ABB RAPID module: Module1.mod

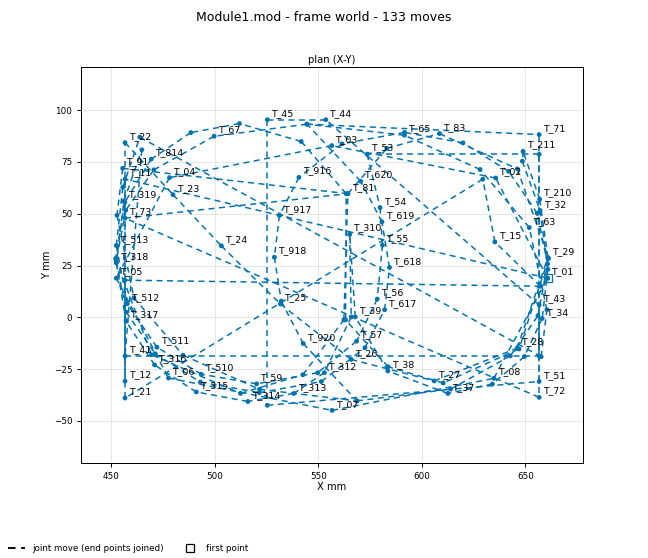
[picture p0: tool path of Module1.mod in frame world, 133 of 133 moves have a stored position in this frame; points joined in program order, loops and branches not executed]
MODULE Module1
    TASK PERS wobjdata Workobject_1:=[FALSE,TRUE,"",[[350,-300,410],[0,0,1,0]],[[0,0,0],[1,0,0,0]]];
    !Zero points
    CONST robtarget T_01:=[[-310.742,318.894,0],[1,0,0,0],[0,0,0,0],[9E+09,9E+09,9E+09,9E+09,9E+09,9E+09]];
    CONST robtarget T_02:=[[-285.702,367.273,0],[1,0,0,0],[0,0,0,0],[9E+09,9E+09,9E+09,9E+09,9E+09,9E+09]];
    CONST robtarget T_03:=[[-206.529,382.913,0],[1,0,0,0],[0,0,0,0],[9E+09,9E+09,9E+09,9E+09,9E+09,9E+09]];
    CONST robtarget T_04:=[[-128.165,367.435,0],[1,0,0,0],[0,0,0,0],[9E+09,9E+09,9E+09,9E+09,9E+09,9E+09]];
    CONST robtarget T_05:=[[-102.477,318.894,0],[1,0,0,0],[0,0,0,0],[9E+09,9E+09,9E+09,9E+09,9E+09,9E+09]];
    CONST robtarget T_06:=[[-127.679,270.676,0],[1,0,0,0],[0,0,0,0],[9E+09,9E+09,9E+09,9E+09,9E+09,9E+09]];
    CONST robtarget T_07:=[[-206.691,255.036,0],[1,0,0,0],[0,0,0,0],[9E+09,9E+09,9E+09,9E+09,9E+09,9E+09]];
    CONST robtarget T_08:=[[-284.811,270.514,0],[1,0,0,0],[0,0,0,0],[9E+09,9E+09,9E+09,9E+09,9E+09,9E+09]];
    CONST robtarget T_09:=[[-310.742,318.894,0],[1,0,0,0],[0,0,0,0],[9E+09,9E+09,9E+09,9E+09,9E+09,9E+09]];
    !One points
    CONST robtarget T_11:=[[-106.691,366.707,0],[1,0,0,0],[0,0,0,0],[9E+09,9E+09,9E+09,9E+09,9E+09,9E+09]];
    CONST robtarget T_12:=[[-106.691,269.138,0],[1,0,0,0],[0,0,0,0],[9E+09,9E+09,9E+09,9E+09,9E+09,9E+09]];
    CONST robtarget T_13:=[[-106.691,317.923,0],[1,0,0,0],[0,0,0,0],[9E+09,9E+09,9E+09,9E+09,9E+09,9E+09]];
    CONST robtarget T_14:=[[-307.339,315.005,0],[1,0,0,0],[0,0,0,0],[9E+09,9E+09,9E+09,9E+09,9E+09,9E+09]];
    CONST robtarget T_15:=[[-285.297,336.399,0],[1,0,0,0],[0,0,0,0],[9E+09,9E+09,9E+09,9E+09,9E+09,9E+09]];
    CONST robtarget T_16:=[[-279.462,366.707,0],[1,0,0,0],[0,0,0,0],[9E+09,9E+09,9E+09,9E+09,9E+09,9E+09]];
    !Two points
    CONST robtarget T_21:=[[-106.691,261.009,0],[1,0,0,0],[0,0,0,0],[9E+09,9E+09,9E+09,9E+09,9E+09,9E+09]];
    CONST robtarget T_22:=[[-106.691,384.347,0],[1,0,0,0],[0,0,0,0],[9E+09,9E+09,9E+09,9E+09,9E+09,9E+09]];
    CONST robtarget T_23:=[[-129.867,359.226,0],[1,0,0,0],[0,0,0,0],[9E+09,9E+09,9E+09,9E+09,9E+09,9E+09]];
    CONST robtarget T_24:=[[-153.206,334.509,0],[1,0,0,0],[0,0,0,0],[9E+09,9E+09,9E+09,9E+09,9E+09,9E+09]];
    CONST robtarget T_25:=[[-181.731,306.39,0],[1,0,0,0],[0,0,0,0],[9E+09,9E+09,9E+09,9E+09,9E+09,9E+09]];
    CONST robtarget T_26:=[[-215.929,279.647,0],[1,0,0,0],[0,0,0,0],[9E+09,9E+09,9E+09,9E+09,9E+09,9E+09]];
    CONST robtarget T_27:=[[-255.961,269.274,0],[1,0,0,0],[0,0,0,0],[9E+09,9E+09,9E+09,9E+09,9E+09,9E+09]];
    CONST robtarget T_28:=[[-296.075,285.077,0],[1,0,0,0],[0,0,0,0],[9E+09,9E+09,9E+09,9E+09,9E+09,9E+09]];
    CONST robtarget T_29:=[[-310.905,328.918,0],[1,0,0,0],[0,0,0,0],[9E+09,9E+09,9E+09,9E+09,9E+09,9E+09]];
    CONST robtarget T_210:=[[-306.934,357.038,0],[1,0,0,0],[0,0,0,0],[9E+09,9E+09,9E+09,9E+09,9E+09,9E+09]];
    CONST robtarget T_211:=[[-298.911,380.133,0],[1,0,0,0],[0,0,0,0],[9E+09,9E+09,9E+09,9E+09,9E+09,9E+09]];
    !Three points
    CONST robtarget T_31:=[[-298.587,375.377,0],[1,0,0,0],[0,0,0,0],[9E+09,9E+09,9E+09,9E+09,9E+09,9E+09]];
    CONST robtarget T_32:=[[-307.096,351.633,0],[1,0,0,0],[0,0,0,0],[9E+09,9E+09,9E+09,9E+09,9E+09,9E+09]];
    CONST robtarget T_33:=[[-310.905,323.189,0],[1,0,0,0],[0,0,0,0],[9E+09,9E+09,9E+09,9E+09,9E+09,9E+09]];
    CONST robtarget T_34:=[[-308.149,299.445,0],[1,0,0,0],[0,0,0,0],[9E+09,9E+09,9E+09,9E+09,9E+09,9E+09]];
    CONST robtarget T_35:=[[-299.559,281.049,0],[1,0,0,0],[0,0,0,0],[9E+09,9E+09,9E+09,9E+09,9E+09,9E+09]];
    CONST robtarget T_36:=[[-284.081,267.759,0],[1,0,0,0],[0,0,0,0],[9E+09,9E+09,9E+09,9E+09,9E+09,9E+09]];
    CONST robtarget T_37:=[[-262.606,263.221,0],[1,0,0,0],[0,0,0,0],[9E+09,9E+09,9E+09,9E+09,9E+09,9E+09]];
    CONST robtarget T_38:=[[-233.595,274.08,0],[1,0,0,0],[0,0,0,0],[9E+09,9E+09,9E+09,9E+09,9E+09,9E+09]];
    CONST robtarget T_39:=[[-217.874,300.174,0],[1,0,0,0],[0,0,0,0],[9E+09,9E+09,9E+09,9E+09,9E+09,9E+09]];
    CONST robtarget T_310:=[[-215.199,340.044,0],[1,0,0,0],[0,0,0,0],[9E+09,9E+09,9E+09,9E+09,9E+09,9E+09]];
    CONST robtarget T_311:=[[-215.929,300.174,0],[1,0,0,0],[0,0,0,0],[9E+09,9E+09,9E+09,9E+09,9E+09,9E+09]];
    CONST robtarget T_312:=[[-202.963,273.27,0],[1,0,0,0],[0,0,0,0],[9E+09,9E+09,9E+09,9E+09,9E+09,9E+09]];
    CONST robtarget T_313:=[[-188.214,263.221,0],[1,0,0,0],[0,0,0,0],[9E+09,9E+09,9E+09,9E+09,9E+09,9E+09]];
    CONST robtarget T_314:=[[-166.01,259.331,0],[1,0,0,0],[0,0,0,0],[9E+09,9E+09,9E+09,9E+09,9E+09,9E+09]];
    CONST robtarget T_315:=[[-141.131,263.95,0],[1,0,0,0],[0,0,0,0],[9E+09,9E+09,9E+09,9E+09,9E+09,9E+09]];
    CONST robtarget T_316:=[[-120.953,276.997,0],[1,0,0,0],[0,0,0,0],[9E+09,9E+09,9E+09,9E+09,9E+09,9E+09]];
    CONST robtarget T_317:=[[-107.177,298.148,0],[1,0,0,0],[0,0,0,0],[9E+09,9E+09,9E+09,9E+09,9E+09,9E+09]];
    CONST robtarget T_318:=[[-102.477,326.268,0],[1,0,0,0],[0,0,0,0],[9E+09,9E+09,9E+09,9E+09,9E+09,9E+09]];
    CONST robtarget T_319:=[[-106.123,356.09,0],[1,0,0,0],[0,0,0,0],[9E+09,9E+09,9E+09,9E+09,9E+09,9E+09]];
    CONST robtarget T_320:=[[-114.794,380.887,0],[1,0,0,0],[0,0,0,0],[9E+09,9E+09,9E+09,9E+09,9E+09,9E+09]];
    !Four points
    CONST robtarget T_41:=[[-106.691,281.323,0],[1,0,0,0],[0,0,0,0],[9E+09,9E+09,9E+09,9E+09,9E+09,9E+09]];
    CONST robtarget T_42:=[[-306.691,281.323,0],[1,0,0,0],[0,0,0,0],[9E+09,9E+09,9E+09,9E+09,9E+09,9E+09]];
    CONST robtarget T_43:=[[-306.691,305.958,0],[1,0,0,0],[0,0,0,0],[9E+09,9E+09,9E+09,9E+09,9E+09,9E+09]];
    CONST robtarget T_44:=[[-203.611,395.424,0],[1,0,0,0],[0,0,0,0],[9E+09,9E+09,9E+09,9E+09,9E+09,9E+09]];
    CONST robtarget T_45:=[[-175.41,395.424,0],[1,0,0,0],[0,0,0,0],[9E+09,9E+09,9E+09,9E+09,9E+09,9E+09]];
    CONST robtarget T_46:=[[-175.41,257.498,0],[1,0,0,0],[0,0,0,0],[9E+09,9E+09,9E+09,9E+09,9E+09,9E+09]];
    !Five points
    CONST robtarget T_51:=[[-306.691,269.007,0],[1,0,0,0],[0,0,0,0],[9E+09,9E+09,9E+09,9E+09,9E+09,9E+09]];
    CONST robtarget T_52:=[[-306.691,378.732,0],[1,0,0,0],[0,0,0,0],[9E+09,9E+09,9E+09,9E+09,9E+09,9E+09]];
    CONST robtarget T_53:=[[-223.611,378.732,0],[1,0,0,0],[0,0,0,0],[9E+09,9E+09,9E+09,9E+09,9E+09,9E+09]];
    CONST robtarget T_54:=[[-229.867,352.962,0],[1,0,0,0],[0,0,0,0],[9E+09,9E+09,9E+09,9E+09,9E+09,9E+09]];
    CONST robtarget T_55:=[[-231.002,334.809,0],[1,0,0,0],[0,0,0,0],[9E+09,9E+09,9E+09,9E+09,9E+09,9E+09]];
    CONST robtarget T_56:=[[-228.49,308.796,0],[1,0,0,0],[0,0,0,0],[9E+09,9E+09,9E+09,9E+09,9E+09,9E+09]];
    CONST robtarget T_57:=[[-218.522,288.456,0],[1,0,0,0],[0,0,0,0],[9E+09,9E+09,9E+09,9E+09,9E+09,9E+09]];
    CONST robtarget T_58:=[[-199.721,273.221,0],[1,0,0,0],[0,0,0,0],[9E+09,9E+09,9E+09,9E+09,9E+09,9E+09]];
    CONST robtarget T_59:=[[-170.224,267.873,0],[1,0,0,0],[0,0,0,0],[9E+09,9E+09,9E+09,9E+09,9E+09,9E+09]];
    CONST robtarget T_510:=[[-143.482,272.492,0],[1,0,0,0],[0,0,0,0],[9E+09,9E+09,9E+09,9E+09,9E+09,9E+09]];
    CONST robtarget T_511:=[[-122.088,285.539,0],[1,0,0,0],[0,0,0,0],[9E+09,9E+09,9E+09,9E+09,9E+09,9E+09]];
    CONST robtarget T_512:=[[-107.744,306.527,0],[1,0,0,0],[0,0,0,0],[9E+09,9E+09,9E+09,9E+09,9E+09,9E+09]];
    CONST robtarget T_513:=[[-102.477,334.647,0],[1,0,0,0],[0,0,0,0],[9E+09,9E+09,9E+09,9E+09,9E+09,9E+09]];
    CONST robtarget T_514:=[[-105.637,362.848,0],[1,0,0,0],[0,0,0,0],[9E+09,9E+09,9E+09,9E+09,9E+09,9E+09]];
    CONST robtarget T_515:=[[-113.822,386.997,0],[1,0,0,0],[0,0,0,0],[9E+09,9E+09,9E+09,9E+09,9E+09,9E+09]];
    !Six points
    CONST robtarget T_61:=[[-307.663,280.947,0],[1,0,0,0],[0,0,0,0],[9E+09,9E+09,9E+09,9E+09,9E+09,9E+09]];
    CONST robtarget T_62:=[[-310.418,303.638,0],[1,0,0,0],[0,0,0,0],[9E+09,9E+09,9E+09,9E+09,9E+09,9E+09]];
    CONST robtarget T_63:=[[-301.909,343.346,0],[1,0,0,0],[0,0,0,0],[9E+09,9E+09,9E+09,9E+09,9E+09,9E+09]];
    CONST robtarget T_64:=[[-278.165,371.385,0],[1,0,0,0],[0,0,0,0],[9E+09,9E+09,9E+09,9E+09,9E+09,9E+09]];
    CONST robtarget T_65:=[[-241.618,387.916,0],[1,0,0,0],[0,0,0,0],[9E+09,9E+09,9E+09,9E+09,9E+09,9E+09]];
    CONST robtarget T_66:=[[-194.535,393.265,0],[1,0,0,0],[0,0,0,0],[9E+09,9E+09,9E+09,9E+09,9E+09,9E+09]];
    CONST robtarget T_67:=[[-149.721,387.43,0],[1,0,0,0],[0,0,0,0],[9E+09,9E+09,9E+09,9E+09,9E+09,9E+09]];
    CONST robtarget T_68:=[[-120.629,371.223,0],[1,0,0,0],[0,0,0,0],[9E+09,9E+09,9E+09,9E+09,9E+09,9E+09]];
    CONST robtarget T_69:=[[-107.015,351.693,0],[1,0,0,0],[0,0,0,0],[9E+09,9E+09,9E+09,9E+09,9E+09,9E+09]];
    CONST robtarget T_610:=[[-102.477,327.138,0],[1,0,0,0],[0,0,0,0],[9E+09,9E+09,9E+09,9E+09,9E+09,9E+09]];
    CONST robtarget T_611:=[[-107.258,302.503,0],[1,0,0,0],[0,0,0,0],[9E+09,9E+09,9E+09,9E+09,9E+09,9E+09]];
    CONST robtarget T_612:=[[-121.277,282.406,0],[1,0,0,0],[0,0,0,0],[9E+09,9E+09,9E+09,9E+09,9E+09,9E+09]];
    CONST robtarget T_613:=[[-143.076,268.71,0],[1,0,0,0],[0,0,0,0],[9E+09,9E+09,9E+09,9E+09,9E+09,9E+09]];
    CONST robtarget T_614:=[[-171.52,263.605,0],[1,0,0,0],[0,0,0,0],[9E+09,9E+09,9E+09,9E+09,9E+09,9E+09]];
    CONST robtarget T_615:=[[-201.504,268.954,0],[1,0,0,0],[0,0,0,0],[9E+09,9E+09,9E+09,9E+09,9E+09,9E+09]];
    CONST robtarget T_616:=[[-222.574,285.323,0],[1,0,0,0],[0,0,0,0],[9E+09,9E+09,9E+09,9E+09,9E+09,9E+09]];
    CONST robtarget T_617:=[[-232.055,303.638,0],[1,0,0,0],[0,0,0,0],[9E+09,9E+09,9E+09,9E+09,9E+09,9E+09]];
    CONST robtarget T_618:=[[-234.405,324.059,0],[1,0,0,0],[0,0,0,0],[9E+09,9E+09,9E+09,9E+09,9E+09,9E+09]];
    CONST robtarget T_619:=[[-230.759,346.101,0],[1,0,0,0],[0,0,0,0],[9E+09,9E+09,9E+09,9E+09,9E+09,9E+09]];
    CONST robtarget T_620:=[[-220.467,365.712,0],[1,0,0,0],[0,0,0,0],[9E+09,9E+09,9E+09,9E+09,9E+09,9E+09]];
    CONST robtarget T_621:=[[-194.535,393.265,0],[1,0,0,0],[0,0,0,0],[9E+09,9E+09,9E+09,9E+09,9E+09,9E+09]];
    !Seven points
    CONST robtarget T_71:=[[-306.691,388.239,0],[1,0,0,0],[0,0,0,0],[9E+09,9E+09,9E+09,9E+09,9E+09,9E+09]];
    CONST robtarget T_72:=[[-306.691,261.334,0],[1,0,0,0],[0,0,0,0],[9E+09,9E+09,9E+09,9E+09,9E+09,9E+09]];
    CONST robtarget T_73:=[[-106.691,347.882,0],[1,0,0,0],[0,0,0,0],[9E+09,9E+09,9E+09,9E+09,9E+09,9E+09]];
    !Eight points
    CONST robtarget T_81:=[[-214.308,359.688,0],[1,0,0,0],[0,0,0,0],[9E+09,9E+09,9E+09,9E+09,9E+09,9E+09]];
    CONST robtarget T_82:=[[-233.109,381.568,0],[1,0,0,0],[-1,0,-1,0],[9E+09,9E+09,9E+09,9E+09,9E+09,9E+09]];
    CONST robtarget T_83:=[[-258.554,388.699,0],[1,0,0,0],[-1,0,-1,0],[9E+09,9E+09,9E+09,9E+09,9E+09,9E+09]];
    CONST robtarget T_84:=[[-296.156,371.681,0],[1,0,0,0],[-1,0,-1,0],[9E+09,9E+09,9E+09,9E+09,9E+09,9E+09]];
    CONST robtarget T_85:=[[-311.229,328.407,0],[1,0,0,0],[-1,0,-1,0],[9E+09,9E+09,9E+09,9E+09,9E+09,9E+09]];
    CONST robtarget T_86:=[[-296.966,284.728,0],[1,0,0,0],[-1,0,-1,0],[9E+09,9E+09,9E+09,9E+09,9E+09,9E+09]];
    CONST robtarget T_87:=[[-260.337,268.278,0],[1,0,0,0],[-1,0,-1,0],[9E+09,9E+09,9E+09,9E+09,9E+09,9E+09]];
    CONST robtarget T_88:=[[-233.757,276.138,0],[1,0,0,0],[-1,0,-1,0],[9E+09,9E+09,9E+09,9E+09,9E+09,9E+09]];
    CONST robtarget T_89:=[[-213.174,298.748,0],[1,0,0,0],[-1,0,-1,0],[9E+09,9E+09,9E+09,9E+09,9E+09,9E+09]];
    CONST robtarget T_810:=[[-213.498,359.688,0],[1,0,0,0],[-1,0,-1,0],[9E+09,9E+09,9E+09,9E+09,9E+09,9E+09]];
    CONST robtarget T_811:=[[-191.78,384.89,0],[1,0,0,0],[-1,0,-1,0],[9E+09,9E+09,9E+09,9E+09,9E+09,9E+09]];
    CONST robtarget T_812:=[[-161.958,393.561,0],[1,0,0,0],[-1,0,-1,0],[9E+09,9E+09,9E+09,9E+09,9E+09,9E+09]];
    CONST robtarget T_813:=[[-138.457,389.185,0],[1,0,0,0],[-1,0,-1,0],[9E+09,9E+09,9E+09,9E+09,9E+09,9E+09]];
    CONST robtarget T_814:=[[-119.332,376.381,0],[1,0,0,0],[-1,0,-1,0],[9E+09,9E+09,9E+09,9E+09,9E+09,9E+09]];
    CONST robtarget T_815:=[[-106.61,355.555,0],[1,0,0,0],[-1,0,-1,0],[9E+09,9E+09,9E+09,9E+09,9E+09,9E+09]];
    CONST robtarget T_816:=[[-102.152,328.407,0],[1,0,0,0],[-1,0,-1,0],[9E+09,9E+09,9E+09,9E+09,9E+09,9E+09]];
    CONST robtarget T_817:=[[-119.494,281.892,0],[1,0,0,0],[0,0,0,0],[9E+09,9E+09,9E+09,9E+09,9E+09,9E+09]];
    CONST robtarget T_818:=[[-162.444,263.253,0],[1,0,0,0],[0,0,0,0],[9E+09,9E+09,9E+09,9E+09,9E+09,9E+09]];
    CONST robtarget T_819:=[[-192.59,272.249,0],[1,0,0,0],[0,0,0,0],[9E+09,9E+09,9E+09,9E+09,9E+09,9E+09]];
    CONST robtarget T_820:=[[-212.363,298.748,0],[1,0,0,0],[0,0,0,0],[9E+09,9E+09,9E+09,9E+09,9E+09,9E+09]];
    CONST robtarget T_821:=[[-214.308,359.688,0],[1,0,0,0],[0,0,0,0],[9E+09,9E+09,9E+09,9E+09,9E+09,9E+09]];
    !Nine points
    CONST robtarget T_91:=[[-105.556,371.949,0],[1,0,0,0],[0,0,0,0],[9E+09,9E+09,9E+09,9E+09,9E+09,9E+09]];
    CONST robtarget T_92:=[[-102.801,349.258,0],[1,0,0,0],[-1,0,-1,0],[9E+09,9E+09,9E+09,9E+09,9E+09,9E+09]];
    CONST robtarget T_93:=[[-110.986,309.388,0],[1,0,0,0],[-1,0,-1,0],[9E+09,9E+09,9E+09,9E+09,9E+09,9E+09]];
    CONST robtarget T_94:=[[-134.729,281.673,0],[1,0,0,0],[-1,0,-1,0],[9E+09,9E+09,9E+09,9E+09,9E+09,9E+09]];
    CONST robtarget T_95:=[[-171.682,265.223,0],[1,0,0,0],[-1,0,-1,0],[9E+09,9E+09,9E+09,9E+09,9E+09,9E+09]];
    CONST robtarget T_96:=[[-218.684,259.631,0],[1,0,0,0],[-1,0,-1,0],[9E+09,9E+09,9E+09,9E+09,9E+09,9E+09]];
    CONST robtarget T_97:=[[-263.903,265.304,0],[1,0,0,0],[-1,0,-1,0],[9E+09,9E+09,9E+09,9E+09,9E+09,9E+09]];
    CONST robtarget T_98:=[[-292.752,281.349,0],[1,0,0,0],[0,0,0,0],[9E+09,9E+09,9E+09,9E+09,9E+09,9E+09]];
    CONST robtarget T_99:=[[-306.123,300.798,0],[1,0,0,0],[0,0,0,0],[9E+09,9E+09,9E+09,9E+09,9E+09,9E+09]];
    CONST robtarget T_910:=[[-310.742,325.757,0],[1,0,0,0],[0,0,0,0],[9E+09,9E+09,9E+09,9E+09,9E+09,9E+09]];
    CONST robtarget T_911:=[[-305.799,350.15,0],[1,0,0,0],[0,0,0,0],[9E+09,9E+09,9E+09,9E+09,9E+09,9E+09]];
    CONST robtarget T_912:=[[-291.942,370.49,0],[1,0,0,0],[0,0,0,0],[9E+09,9E+09,9E+09,9E+09,9E+09,9E+09]];
    CONST robtarget T_913:=[[-269.9,384.266,0],[1,0,0,0],[0,0,0,0],[9E+09,9E+09,9E+09,9E+09,9E+09,9E+09]];
    CONST robtarget T_914:=[[-241.699,389.291,0],[1,0,0,0],[0,0,0,0],[9E+09,9E+09,9E+09,9E+09,9E+09,9E+09]];
    CONST robtarget T_915:=[[-211.472,383.78,0],[1,0,0,0],[0,0,0,0],[9E+09,9E+09,9E+09,9E+09,9E+09,9E+09]];
    CONST robtarget T_916:=[[-190.645,367.573,0],[1,0,0,0],[0,0,0,0],[9E+09,9E+09,9E+09,9E+09,9E+09,9E+09]];
    CONST robtarget T_917:=[[-181.245,349.177,0],[1,0,0,0],[0,0,0,0],[9E+09,9E+09,9E+09,9E+09,9E+09,9E+09]];
    CONST robtarget T_918:=[[-178.814,328.999,0],[1,0,0,0],[0,0,0,0],[9E+09,9E+09,9E+09,9E+09,9E+09,9E+09]];
    CONST robtarget T_919:=[[-182.136,307.767,0],[1,0,0,0],[0,0,0,0],[9E+09,9E+09,9E+09,9E+09,9E+09,9E+09]];
    CONST robtarget T_920:=[[-192.752,287.346,0],[1,0,0,0],[0,0,0,0],[9E+09,9E+09,9E+09,9E+09,9E+09,9E+09]];
    CONST robtarget T_921:=[[-218.684,259.631,0],[1,0,0,0],[0,0,0,0],[9E+09,9E+09,9E+09,9E+09,9E+09,9E+09]];
    PROC Path_10()
        MoveJ T_01,v100,z10,VacuumGripper\WObj:=Workobject_1;
        MoveJ T_02,v100,z10,VacuumGripper\WObj:=Workobject_1;
        MoveJ T_03,v100,z10,VacuumGripper\WObj:=Workobject_1;
        MoveJ T_04,v100,z10,VacuumGripper\WObj:=Workobject_1;
        MoveJ T_05,v100,z10,VacuumGripper\WObj:=Workobject_1;
        MoveJ T_06,v100,z10,VacuumGripper\WObj:=Workobject_1;
        MoveJ T_07,v100,z10,VacuumGripper\WObj:=Workobject_1;
        MoveJ T_08,v100,z10,VacuumGripper\WObj:=Workobject_1;
        MoveJ T_09,v100,z10,VacuumGripper\WObj:=Workobject_1;
        MoveJ T_11,v100,z10,VacuumGripper\WObj:=Workobject_1;
        MoveJ T_12,v100,z10,VacuumGripper\WObj:=Workobject_1;
        MoveJ T_13,v100,z10,VacuumGripper\WObj:=Workobject_1;
        MoveJ T_14,v100,z10,VacuumGripper\WObj:=Workobject_1;
        MoveJ T_15,v100,z10,VacuumGripper\WObj:=Workobject_1;
        MoveJ T_16,v100,z10,VacuumGripper\WObj:=Workobject_1;
        MoveJ T_21,v100,z10,VacuumGripper\WObj:=Workobject_1;
        MoveJ T_22,v100,z10,VacuumGripper\WObj:=Workobject_1;
        MoveJ T_23,v100,z10,VacuumGripper\WObj:=Workobject_1;
        MoveJ T_24,v100,z10,VacuumGripper\WObj:=Workobject_1;
        MoveJ T_25,v100,z10,VacuumGripper\WObj:=Workobject_1;
        MoveJ T_26,v100,z10,VacuumGripper\WObj:=Workobject_1;
        MoveJ T_27,v100,z10,VacuumGripper\WObj:=Workobject_1;
        MoveJ T_28,v100,z10,VacuumGripper\WObj:=Workobject_1;
        MoveJ T_29,v100,z10,VacuumGripper\WObj:=Workobject_1;
        MoveJ T_210,v100,z10,VacuumGripper\WObj:=Workobject_1;
        MoveJ T_211,v100,z10,VacuumGripper\WObj:=Workobject_1;
        MoveJ T_31,v100,z10,VacuumGripper\WObj:=Workobject_1;
        MoveJ T_32,v100,z10,VacuumGripper\WObj:=Workobject_1;
        MoveJ T_33,v100,z10,VacuumGripper\WObj:=Workobject_1;
        MoveJ T_34,v100,z10,VacuumGripper\WObj:=Workobject_1;
        MoveJ T_35,v100,z10,VacuumGripper\WObj:=Workobject_1;
        MoveJ T_36,v100,z10,VacuumGripper\WObj:=Workobject_1;
        MoveJ T_37,v100,z10,VacuumGripper\WObj:=Workobject_1;
        MoveJ T_38,v100,z10,VacuumGripper\WObj:=Workobject_1;
        MoveJ T_39,v100,z10,VacuumGripper\WObj:=Workobject_1;
        MoveJ T_310,v100,z10,VacuumGripper\WObj:=Workobject_1;
        MoveJ T_311,v100,z10,VacuumGripper\WObj:=Workobject_1;
        MoveJ T_312,v100,z10,VacuumGripper\WObj:=Workobject_1;
        MoveJ T_313,v100,z10,VacuumGripper\WObj:=Workobject_1;
        MoveJ T_314,v100,z10,VacuumGripper\WObj:=Workobject_1;
        MoveJ T_315,v100,z10,VacuumGripper\WObj:=Workobject_1;
        MoveJ T_316,v100,z10,VacuumGripper\WObj:=Workobject_1;
        MoveJ T_317,v100,z10,VacuumGripper\WObj:=Workobject_1;
        MoveJ T_318,v100,z10,VacuumGripper\WObj:=Workobject_1;
        MoveJ T_319,v100,z10,VacuumGripper\WObj:=Workobject_1;
        MoveJ T_320,v100,z10,VacuumGripper\WObj:=Workobject_1;
        MoveJ T_41,v100,z10,VacuumGripper\WObj:=Workobject_1;
        MoveJ T_42,v100,z10,VacuumGripper\WObj:=Workobject_1;
        MoveJ T_43,v100,z10,VacuumGripper\WObj:=Workobject_1;
        MoveJ T_44,v100,z10,VacuumGripper\WObj:=Workobject_1;
        MoveJ T_45,v100,z10,VacuumGripper\WObj:=Workobject_1;
        MoveJ T_46,v100,z10,VacuumGripper\WObj:=Workobject_1;
        MoveJ T_51,v100,z10,VacuumGripper\WObj:=Workobject_1;
        MoveJ T_52,v100,z10,VacuumGripper\WObj:=Workobject_1;
        MoveJ T_53,v100,z10,VacuumGripper\WObj:=Workobject_1;
        MoveJ T_54,v100,z10,VacuumGripper\WObj:=Workobject_1;
        MoveJ T_55,v100,z10,VacuumGripper\WObj:=Workobject_1;
        MoveJ T_56,v100,z10,VacuumGripper\WObj:=Workobject_1;
        MoveJ T_57,v100,z10,VacuumGripper\WObj:=Workobject_1;
        MoveJ T_58,v100,z10,VacuumGripper\WObj:=Workobject_1;
        MoveJ T_59,v100,z10,VacuumGripper\WObj:=Workobject_1;
        MoveJ T_510,v100,z10,VacuumGripper\WObj:=Workobject_1;
        MoveJ T_511,v100,z10,VacuumGripper\WObj:=Workobject_1;
        MoveJ T_512,v100,z10,VacuumGripper\WObj:=Workobject_1;
        MoveJ T_513,v100,z10,VacuumGripper\WObj:=Workobject_1;
        MoveJ T_514,v100,z10,VacuumGripper\WObj:=Workobject_1;
        MoveJ T_515,v100,z10,VacuumGripper\WObj:=Workobject_1;
        MoveJ T_61,v100,z10,VacuumGripper\WObj:=Workobject_1;
        MoveJ T_62,v100,z10,VacuumGripper\WObj:=Workobject_1;
        MoveJ T_63,v100,z10,VacuumGripper\WObj:=Workobject_1;
        MoveJ T_64,v100,z10,VacuumGripper\WObj:=Workobject_1;
        MoveJ T_65,v100,z10,VacuumGripper\WObj:=Workobject_1;
        MoveJ T_66,v100,z10,VacuumGripper\WObj:=Workobject_1;
        MoveJ T_67,v100,z10,VacuumGripper\WObj:=Workobject_1;
        MoveJ T_68,v100,z10,VacuumGripper\WObj:=Workobject_1;
        MoveJ T_69,v100,z10,VacuumGripper\WObj:=Workobject_1;
        MoveJ T_610,v100,z10,VacuumGripper\WObj:=Workobject_1;
        MoveJ T_611,v100,z10,VacuumGripper\WObj:=Workobject_1;
        MoveJ T_612,v100,z10,VacuumGripper\WObj:=Workobject_1;
        MoveJ T_613,v100,z10,VacuumGripper\WObj:=Workobject_1;
        MoveJ T_614,v100,z10,VacuumGripper\WObj:=Workobject_1;
        MoveJ T_615,v100,z10,VacuumGripper\WObj:=Workobject_1;
        MoveJ T_616,v100,z10,VacuumGripper\WObj:=Workobject_1;
        MoveJ T_617,v100,z10,VacuumGripper\WObj:=Workobject_1;
        MoveJ T_618,v100,z10,VacuumGripper\WObj:=Workobject_1;
        MoveJ T_619,v100,z10,VacuumGripper\WObj:=Workobject_1;
        MoveJ T_620,v100,z10,VacuumGripper\WObj:=Workobject_1;
        MoveJ T_621,v100,z10,VacuumGripper\WObj:=Workobject_1;
        MoveJ T_71,v100,z10,VacuumGripper\WObj:=Workobject_1;
        MoveJ T_72,v100,z10,VacuumGripper\WObj:=Workobject_1;
        MoveJ T_73,v100,z10,VacuumGripper\WObj:=Workobject_1;
        MoveJ T_81,v100,z10,VacuumGripper\WObj:=Workobject_1;
        MoveJ T_82,v100,z10,VacuumGripper\WObj:=Workobject_1;
        MoveJ T_83,v100,z10,VacuumGripper\WObj:=Workobject_1;
        MoveJ T_84,v100,z10,VacuumGripper\WObj:=Workobject_1;
        MoveJ T_85,v100,z10,VacuumGripper\WObj:=Workobject_1;
        MoveJ T_86,v100,z10,VacuumGripper\WObj:=Workobject_1;
        MoveJ T_87,v100,z10,VacuumGripper\WObj:=Workobject_1;
        MoveJ T_88,v100,z10,VacuumGripper\WObj:=Workobject_1;
        MoveJ T_89,v100,z10,VacuumGripper\WObj:=Workobject_1;
        MoveJ T_810,v100,z10,VacuumGripper\WObj:=Workobject_1;
        MoveJ T_811,v100,z10,VacuumGripper\WObj:=Workobject_1;
        MoveJ T_812,v100,z10,VacuumGripper\WObj:=Workobject_1;
        MoveJ T_813,v100,z10,VacuumGripper\WObj:=Workobject_1;
        MoveJ T_814,v100,z10,VacuumGripper\WObj:=Workobject_1;
        MoveJ T_815,v100,z10,VacuumGripper\WObj:=Workobject_1;
        MoveJ T_816,v100,z10,VacuumGripper\WObj:=Workobject_1;
        MoveJ T_817,v100,z10,VacuumGripper\WObj:=Workobject_1;
        MoveJ T_818,v100,z10,VacuumGripper\WObj:=Workobject_1;
        MoveJ T_819,v100,z10,VacuumGripper\WObj:=Workobject_1;
        MoveJ T_820,v100,z10,VacuumGripper\WObj:=Workobject_1;
        MoveJ T_821,v100,z10,VacuumGripper\WObj:=Workobject_1;
        MoveJ T_91,v100,z10,VacuumGripper\WObj:=Workobject_1;
        MoveJ T_92,v100,z10,VacuumGripper\WObj:=Workobject_1;
        MoveJ T_93,v100,z10,VacuumGripper\WObj:=Workobject_1;
        MoveJ T_94,v100,z10,VacuumGripper\WObj:=Workobject_1;
        MoveJ T_95,v100,z10,VacuumGripper\WObj:=Workobject_1;
        MoveJ T_96,v100,z10,VacuumGripper\WObj:=Workobject_1;
        MoveJ T_97,v100,z10,VacuumGripper\WObj:=Workobject_1;
        MoveJ T_98,v100,z10,VacuumGripper\WObj:=Workobject_1;
        MoveJ T_99,v100,z10,VacuumGripper\WObj:=Workobject_1;
        MoveJ T_910,v100,z10,VacuumGripper\WObj:=Workobject_1;
        MoveJ T_911,v100,z10,VacuumGripper\WObj:=Workobject_1;
        MoveJ T_912,v100,z10,VacuumGripper\WObj:=Workobject_1;
        MoveJ T_913,v100,z10,VacuumGripper\WObj:=Workobject_1;
        MoveJ T_914,v100,z10,VacuumGripper\WObj:=Workobject_1;
        MoveJ T_915,v100,z10,VacuumGripper\WObj:=Workobject_1;
        MoveJ T_916,v100,z10,VacuumGripper\WObj:=Workobject_1;
        MoveJ T_917,v100,z10,VacuumGripper\WObj:=Workobject_1;
        MoveJ T_918,v100,z10,VacuumGripper\WObj:=Workobject_1;
        MoveJ T_919,v100,z10,VacuumGripper\WObj:=Workobject_1;
        MoveJ T_920,v100,z10,VacuumGripper\WObj:=Workobject_1;
        MoveJ T_921,v100,z10,VacuumGripper\WObj:=Workobject_1;
    ENDPROC
ENDMODULE
